{attribute 'linkalways'} 
{attribute 'no_explicit_call' := 'This FB is a CLASS and must be accessed using methods or properties'}
{attribute 'enable_dynamic_creation'}
FUNCTION_BLOCK ABSTRACT DefaultDisposable IMPLEMENTS Disposable

METHOD PUBLIC Dispose
VAR
	pDisposable : POINTER TO DefaultDisposable;
END_VAR
pDisposable := THIS;
__DELETE(pDisposable);
END_METHOD

METHOD FB_exit : BOOL
VAR_INPUT
	bInCopyCode : BOOL; // if TRUE, the exit method is called for exiting an instance that is copied afterwards (online change).
END_VAR
// by default you would return if this is an in copy code, i.e. online change to this class
IF bInCopyCode THEN
	RETURN;
END_IF

// A word of warning. FB_exit does not NOT operate in the same way as a typical inherited method. If a child class does not implement FB_exit then it does not
// gain this one for itself. 
// The system will automatically call each FB_exit on each layer of inheritance one by one, starting with the child class and making it's way to the parent.
// Therefore code in here will only be triggered once the system reaches this layer of the object's deletion. The child class and all of it's variables
// will already have had FB_exit called by the time we reach this point!
END_METHOD

END_FUNCTION_BLOCK

(* stored: Version 1.1.0.1
   POU DefaultDisposable: Id {7157366b-07e8-46fc-aa2f-38c2e2eab868}, SpecialFunc None
   Folder Destructor: Id {a244c56d-214c-0539-02cc-30986d16b566}
   Method Dispose: Id {6c98f403-5dd6-4f9d-bc0a-e406c48a07a8}
   Method FB_exit: Id {0d1dd945-173c-0626-2abd-474b81e0db04} *)
